// SIMATIC S7-200 project (STEP 7-Micro/WIN), CPU 224XP CN REL 02.01

ORGANIZATION_BLOCK MAIN:OB1
TITLE=PROGRAM COMMENTS
BEGIN
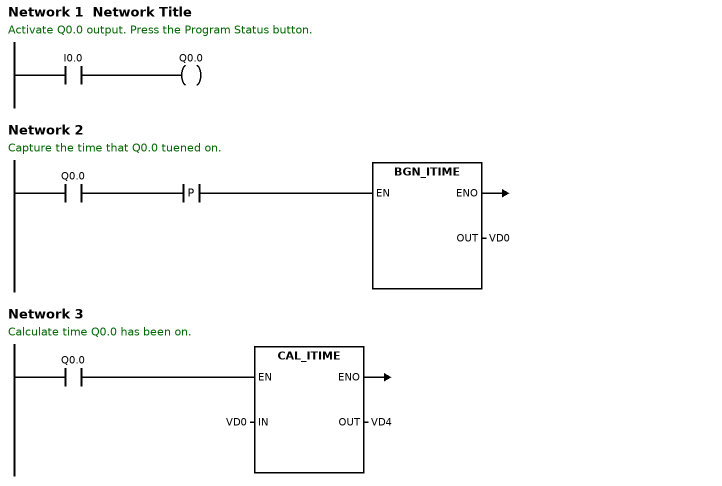
Network 1 // Network Title
// Activate Q0.0 output. Press the Program Status button.
LD     I0.0
=      Q0.0
Network 2
// Capture the time that Q0.0 tuened on.
LD     Q0.0
EU
BITIM  VD0
Network 3
// Calculate time Q0.0 has been on.
LD     Q0.0
CITIM  VD0, VD4
END_ORGANIZATION_BLOCK
